TYPE ST_HMI_C1_Ctrl3_State_Unit : 
STRUCT
	//State_Unit
	bTrigReconfigure: BOOL;
	sM1_sOutput: STRING(255); //Value
END_STRUCT
END_TYPE

(* stored: DUT ST_HMI_C1_Ctrl3_State_Unit: Id ac90f9eb-6b85-4ac6-a37d-714c7691a858 *)
